// TwinCAT 3 PLC project PLC_SelfWrittenFunctionBasics
// ProgramVersion: 3.1.4024.12
// libraries:
//   Tc2_Standard, * (Beckhoff Automation GmbH)
//   Tc2_System, * (Beckhoff Automation GmbH)
//   Tc3_Module, * (Beckhoff Automation GmbH)
//   Tc3_Vision, * (Beckhoff Automation GmbH)
// project tree:
//   / PlcTask.TcTTO
//   POUs/ F_CountAndDrawObjects.TcPOU, MAIN.TcPOU
// real-time tasks:
//   TASK PlcTask: cycle T#10ms, priority 20, ADS port 350
//   TASK VnTask ImgAcq (FileSource1): cycle T#10ms, priority 5, ADS port 351

CONFIGURATION PLC_SelfWrittenFunctionBasics
    RESOURCE PLC ON TwinCAT3
        TASK PlcTask(INTERVAL := T#10ms, PRIORITY := 20);
        PROGRAM MAIN WITH PlcTask : MAIN;
    END_RESOURCE
END_CONFIGURATION

// ---- POUs/MAIN.TcPOU
PROGRAM MAIN
VAR
	hr				:	HRESULT;
	fbCameraControl	:	FB_VN_SimpleCameraControl;
	eCameraState	:	ETcVnCameraState;
	
	ipImageIn		:	ITcVnImage;
	ipImageInDisp	:	ITcVnDisplayableImage;
	ipImageRes		:	ITcVnImage;
	ipImageResDisp	:	ITcVnDisplayableImage;
	
	aColorGreen		:	TcVnVector4_LREAL := [0, 255, 0, 0];
	nNumber			:	ULINT;
	sText           :	STRING(255);
END_VAR

//	Disclaimer
  	
//	THIS publication contains statements about the suitability OF our products FOR certain 
//	areas OF application. These statements are based on typical features OF our products. 
//	The examples shown in THIS publication are FOR demonstration purposes only. The 
//	information provided herein should NOT be regarded as specific operation characteristics. 
//	It is incumbent on the customer TO check AND decide whether a product is suitable FOR use 
//	in a particular application. We DO NOT give ANY warranty that the source code which is 
//	made available with this publication is complete or accurate. 
  	
//	THE SAMPLE CODE CONTAINED IN THIS PUBLICATION IS PROVIDED “AS IS” WITHOUT WARRANTY OF ANY 
//	KIND, EITHER EXPRESSED, IMPLIED OR STATUTORY, INCLUDING WITHOUT LIMITATION, ANY WARRANTY 
//	WITH RESPECT TO NON-INFRINGEMENT, FREEDOM FROM PROPRIETARY RIGHTS OF THIRD PARTIES OR 
//	FITNESS FOR ANY PARTICULAR PURPOSE. 
  	
//	THIS publication may be changed FROM TIME TO TIME without prior notice. No liability 
//	is assumed FOR errors AND/OR omissions. Our products are described in detail in our 
//	data sheets AND documentations. Product-specific warnings AND cautions must be observed. 
//	FOR the latest version OF our data sheets AND documentations visit our website 
//	(www.beckhoff.de). 
  	
//	© Beckhoff Automation GmbH & Co. KG, March 2020
  	
//	The reproduction, distribution AND utilization OF THIS document as well as the 
//	communication OF its contents TO others without express authorization is prohibited. 
//	Offenders will be held liable FOR the payment OF damages. All rights reserved in the 
//	event of the grant of a patent, utility model or design.

//	==========================================================================================

//	Sample: Self Written Functions
//	----------------------------------------

//	Steps to do:
//	 1. Add images to the FileSource1

eCameraState := fbCameraControl.GetState();

// CameraControl is in error state, so try to reset the camera connection
IF eCameraState = TCVN_CS_ERROR THEN
	hr := fbCameraControl.Reset();

// Camera not yet streaming
ELSIF eCameraState < TCVN_CS_ACQUIRING THEN
	hr := fbCameraControl.StartAcquisition();

// Camera streaming
ELSIF eCameraState = TCVN_CS_ACQUIRING THEN
	hr := fbCameraControl.GetCurrentImage(ipImageIn);
	
	IF SUCCEEDED(hr) AND ipImageIn <> 0 THEN
		// Do stuff…
		hr := F_CountAndDrawObjects(ipImageIn, ipImageRes, aColorGreen, nNumber, hr);
		
		// Write Number Result
		sText := CONCAT('Number ', ULINT_TO_STRING(nNumber));
		hr := F_VN_PutTextExp(sText, ipImageRes, 25, 50, TCVN_FT_HERSHEY_SIMPLEX, 1.3, aColorGreen, 2, TCVN_LT_8_CONNECTED, FALSE,hr);
		
		// Display Images
		hr := F_VN_TransformIntoDisplayableImage(ipImageIn, ipImageInDisp, hr);
		hr := F_VN_TransformIntoDisplayableImage(ipImageRes, ipImageResDisp, hr);
	END_IF
END_IF

END_PROGRAM

// ---- POUs/F_CountAndDrawObjects.TcPOU
FUNCTION F_CountAndDrawObjects : HRESULT
VAR_INPUT
	ipSrcImage			:	ITcVnImage;
	ipDestImage			:	REFERENCE TO ITcVnImage;
	aColor				:	TcVnVector4_LREAL;
	nNumberOfObjects	:	REFERENCE TO ULINT;
	hrPrev				:	HRESULT;
END_VAR
VAR
	hr					:	HRESULT;
	ipContours			:	ITcVnContainer;
	stParams			:	TcVnParamsBlobDetection;
END_VAR

// Check previous HRESULT
// Skip this function, if previous functions failed
IF FAILED(hrPrev) THEN
	F_CountAndDrawObjects := hrPrev;
	RETURN;
END_IF

// Check if all the interface pointer in VAR_INPUT are valid (here: ipSrcImage)
// Otherwise return INVALIDPARM and skip function
IF ipSrcImage = 0 THEN
	F_CountAndDrawObjects := Tc2_System.E_HRESULTAdsErr.INVALIDPARM;
	RETURN;
END_IF

// Examplary vision functionality
hr := F_VN_ConvertColorSpace(ipSrcImage, ipDestImage, TCVN_CST_GRAY_TO_RGB, hr);
stParams.bFilterByArea := TRUE;
stParams.fMinArea := 10_000;
stParams.fMaxArea := 100_000;
hr := F_VN_DetectBlobs(ipSrcImage, ipContours, stParams, hr);
hr := F_VN_GetNumberOfElements(ipContours, nNumberOfObjects, hr);
hr := F_VN_DrawContours(ipContours, -1, ipDestImage, aColor, 5, hr);

// Release all interface pointers declared in this function
FW_SafeRelease(ADR(ipContours));

// Return the HRESULT
F_CountAndDrawObjects := hr;

END_FUNCTION
